TYPE ST_HMI_BASE_STATION_MANUAL_IN :
STRUCT
	diSelectedObjectIndex	: DINT;
	stControl				: ST_HMI_GRID_IN;
	stManualCylinder		: ST_HMI_MANUAL_CYLINDER_IN;
	stManualDrive			: ST_HMI_MANUAL_DRIVE_IN;
	stManualAxis			: ST_HMI_MANUAL_AXIS_IN;
	stManualDevice			: ST_HMI_MANUAL_DEVICE_IN;	
END_STRUCT
END_TYPE

(* stored: Version 1.1.0.1, ProductVersion 3.1.4024.12
   DUT ST_HMI_BASE_STATION_MANUAL_IN: Id {94e20563-b986-4810-8acb-bbb2f7f36094} *)
